// TIA Portal V17 export
// export: Created 2025-03-07T09:18:23.4469488Z, ExportSetting WithDefaults, DisplayName Totally Integrated Automation Portal, DisplayVersion V17 Update 8, DisplayName TIA Portal Openness, DisplayVersion V17 Update 8, DisplayName TIA Portal Version Control Interface, DisplayVersion V17, DisplayName SINAMICS Startdrive Advanced, DisplayVersion V17 SP2, DisplayName SINAMICS Startdrive G110M, G120, G120C, G120D, G120P, G115D, DisplayVersion V17 SP2, DisplayName SINAMICS Startdrive G130, G150, S120, S150, SINAMICS MV, S210, DisplayVersion V17 SP2, DisplayName STEP 7 Professional, DisplayVersion V17 Update 8, DisplayName SINUMERIK ONE STEP 7 Toolbox, DisplayVersion V17 Update 12, DisplayName SINUMERIK 840D sl STEP 7 Toolbox, DisplayVersion V17 Update 12, DisplayName STEP 7 Safety, DisplayVersion V17 Update 6, DisplayName WinCC Advanced, DisplayVersion V17 Update 8
FUNCTION_BLOCK "FB1453_LASER_COOLING_ALARMS"   // FB1453, LAD
{ S7_Optimized_Access := 'FALSE' }
AUTHOR : ETXETAR
VERSION : 1.0
// stored: AutoNumber false, IsIECCheckEnabled false, SetENOAutomatically false, UDAEnableTagReadback false
   VAR_INPUT
      OPTIONS_0 : Byte := 2#0000_0000;   // OPTIONS 0
      OPTIONS_1 : Byte := 2#0000_0000;   // OPTIONS 1
      LASER_OUTPUT_FLOW_LOW_VALUE_ALM_BIT : Bool;   // LASER OUTPUT FLOW LOW LEVEL ALARM BIT INPUT
      NOZZLE_FLOW_LOW_VALUE_ALM_BIT : Bool;   // NOZZLE FLOW LOW LEVEL ALARM BIT INPUT
      HEAD_FLOW_LOW_VALUE_ALM_BIT : Bool;   // HEAD FLOW LOW LEVEL ALARM BIT INPUT
      LASER_OUTPUT_OVERTEMPERATURE_ALM_BIT : Bool;   // LASER OUTPUT OVERTEMPERATURE ALARM BIT INPUT
      NOZZLE_OVERTEMPERATURE_ALM_BIT : Bool;   // NOZZLE OVERTEMPERATURE ALARM BIT INPUT
      HEAD_OVERTEMPERATURE_ALM_BIT : Bool;   // HEAD OVERTEMPERATURE ALARM BIT INPUT
      LASER_OUTPUT_FLOW_RAW_INPUT : DInt;   // LASER OUTPUT FLOW RAW INPUT
      LASER_OUTPUT_TEMP_RAW_INPUT : DInt;   // LASER OUTPUT TEMPERATURE RAW INPUT
      NOZZLE_COOLING_FLOW_RAW_INPUT : Word;   // NOZZLE FLOW RAW INPUT
      NOZZLE_COOLING_TEMP_RAW_INPUT : Word;   // NOOZLE TEMPERATURE RAW INPUT
      HEAD_COOLING_FLOW_RAW_INPUT : DInt;   // HEAD FLOW RAW INPUT
      HEAD_COOLING_TEMP_RAW_INPUT : DInt;   // HEAD TEMPERATURE RAW INPUT
      LASER_READY : Bool;   // THE LASER DEVICE IS READY
      UNIT_ALARM : UInt;   // UNIT NUMBER MAX. NUMBER=10
   END_VAR
   VAR_OUTPUT
      OUTPUT_LOW_FLOW_ALARM : Bool;   // LASER OUTPUT COOLING LOW FLOW ALARM
      OUTPUT_HIGH_FLOW_ALARM : Bool;   // LASER OUTPUT COOLING HIGH FLOW ALARM
      OUTPUT_FLOW_SETPOINT_ALARM : Bool;   // LASER OUTPUT COOLING FLOW SETPOINT ALARM
      OUTPUT_LOW_TEMP_ALARM : Bool;   // LASER OUTPUT COOLING LOW TEMPERATURE ALARM
      OUTPUT_HIGH_TEMP_ALARM : Bool;   // LASER OUTPUT COOLING HIGH TEMPERATURE ALARM
      OUTPUT_TEMP_SETPOINT_ALARM : Bool;   // LASER OUTPUT COOLING TEMPERATURE SETPOINT ALARM
      NOZZLE_LOW_FLOW_ALARM : Bool;   // NOZZLE COOLING LOW FLOW ALARM
      NOZZLE_HIGH_FLOW_ALARM : Bool;   // NOZZLE COOLING HIGH FLOW ALARM
      NOZZLE_FLOW_SETPOINT_ALARM : Bool;   // NOZZLE COOLING FLOW SETPOINT ALARM
      NOZZLE_LOW_TEMP_ALARM : Bool;   // NOZZLE COOLING LOW TEMPERATURE ALARM
      NOZZLE_HIGH_TEMP_ALARM : Bool;   // NOZZLE COOLING HIGH TEMPERATURE ALARM
      NOZZLE_TEMP_SETPOINT_ALARM : Bool;   // NOZZLE COOLING TEMPERATURE SETPOINT ALARM
      HEAD_LOW_FLOW_ALARM : Bool;   // LASER HEAD COOLING LOW FLOW ALARM
      HEAD_HIGH_FLOW_ALARM : Bool;   // LASER HEAD COOLING HIGH FLOW ALARM
      HEAD_FLOW_SETPOINT_ALARM : Bool;   // LASER HEAD COOLING FLOW SETPOINT ALARM
      HEAD_LOW_TEMP_ALARM : Bool;   // LASER HEAD COOLING LOW TEMPERATURE ALARM
      HEAD_HIGH_TEMP_ALARM : Bool;   // LASER HEAD COOLING HIGH TEMPERATURE ALARM
      HEAD_TEMP_SETPOINT_ALARM : Bool;   // LASER HEAD COOLING TEMPERATURE SETPOINT ALARM
      OUTPUT_LOW_FLOW_WARNING : Bool;   // LASER OUTPUT COOLING LOW FLOW WARNING
      OUTPUT_HIGH_FLOW_WARNING : Bool;   // LASER OUTPUT COOLING HIGH FLOW WARNING
      OUTPUT_LOW_TEMP_WARNING : Bool;   // LASER OUTPUT COOLING LOW TEMPERATURE WARNING
      OUTPUT_HIGH_TEMP_WARNING : Bool;   // LASER OUTPUT COOLING HIGH TEMPERATURE WARNING
      NOZZLE_LOW_FLOW_WARNING : Bool;   // NOZZLE COOLING LOW FLOW WARNING
      NOZZLE_HIGH_FLOW_WARNING : Bool;   // NOZZLE COOLING HIGH FLOW WARNING
      NOZZLE_LOW_TEMP_WARNING : Bool;   // NOZZLE COOLING LOW TEMPERATURE WARNING
      NOZZLE_HIGH_TEMP_WARNING : Bool;   // NOZZLE COOLING HIGH TEMPERATURE WARNING
      HEAD_LOW_FLOW_WARNING : Bool;   // LASER HEAD COOLING LOW FLOW WARNING
      HEAD_HIGH_FLOW_WARNING : Bool;   // LASER HEAD COOLING HIGH FLOW WARNING
      HEAD_LOW_TEMP_WARNING : Bool;   // LASER HEAD COOLING LOW TEMPERATURE WARNING
      HEAD_HIGH_TEMP_WARNING : Bool;   // LASER HEAD COOLING HIGH TEMPERATURE WARNING
   END_VAR
   VAR DB_SPECIFIC
      ANY_ACTIVE_ALARM : Bool;   // ANY ACTIVE ALARM
      RHP_SEOC_ALARMS : Bool;   // RETURN HOME POSITION AND STOP END OF CYCLE ALARMS
      IS_SEOC_ALARMS : Bool;   // INMEDIATE STOP AND STOP END OF CYCLE ALARMS
      WARNINGS : Bool;   // WARNINGS
      WARNINGS_GONE : Bool;   // WARNINGS GONE
      COOLING_ALARMS_ENABLED : Bool;   // COOLING ALARMS ENABLED
      LASER_OUTPUT_SENSOR_VALUES { ExternalAccessible := 'False'; ExternalVisible := 'False'; ExternalWritable := 'False'} : "COOLING_SENSOR";
      NOZZLE_SENSOR_VALUES { ExternalAccessible := 'False'; ExternalVisible := 'False'; ExternalWritable := 'False'} : "COOLING_SENSOR";
      LASER_HEAD_SENSOR_VALUES { ExternalAccessible := 'False'; ExternalVisible := 'False'; ExternalWritable := 'False'} : "COOLING_SENSOR";
   END_VAR
   VAR_TEMP
      INPUTS_MASK : Byte;   // INPUT MASK
      O_BYTE_0 : Struct   // OPTIONS BYTE 0
         OUTPUT_FLOW_LOW_BIT_ALARM : Bool;   // CIRCUIT BREAKER OPTION
         NOZZLE_FLOW_LOW_BIT_ALARM : Bool;   // CONTACTOR FEEDBACK OPTION
         HEAD_FLOW_LOW_BIT_ALARM : Bool;   // LOW LEVEL ALARM OPTION
         OUTPUT_FLOW_ANALOG_VALUE : Bool;   // SYSTEM ALARM 1 OPTION
         NOZZLE_FLOW_ANALOG_VALUE : Bool;   // SYSTEM ALARM 2 OPTION
         HEAD_FLOW_ANALOG_VALUE : Bool;   // FILTER CLOGGED ALARM OPTION
         SPARE_6 : Bool;   // OVERTEMPERATURE ALARM OPTION
         SPARE_7 : Bool;   // WATER SUPPLY FLOW OPTION
      END_STRUCT;
      O_BYTE_1 : Struct   // OPTIONS BYTE 1
         OUTPUT_TEMP_HIGH_BIT_ALARM : Bool;   // LOW LEVEL PREALARM OPTION
         NOZZLE_TEMP_HIGH_BIT_ALARM : Bool;   // FILTER CLOGGED PREALARM OPTION
         HEAD_TEMP_HIGH_BIT_ALARM : Bool;   // OVERTEMPERATURE PREALARM OPTION
         OUTPUT_TEMP_ANALOG_VALUE : Bool;   // DIGITAL FLOW SENSORS OPTION
         NOZZLE_TEMP_ANALOG_VALUE : Bool;   // SPARE OPTION
         HEAD_TEMP_ANALOG_VALUE : Bool;   // SPARE OPTION
         SPARE_6 : Bool;   // SPARE OPTION
         SPARE_7 : Bool;   // SPARE OPTION
      END_STRUCT;
      DB_NUMBER : DInt;   // DB NUMBER FOR ALARM AND HELP DECODING
      COOLING_TEMP_AUX_OUTPUT : Real;   // COOLING OUTPUT TEMPERATURE AUX
      COOLING_FLOW_AUX_OUTPUT : Real;   // COOLING OUTPUT FLOW AUX
      COOLING_TEMP_AUX_3 : Int;   // COOLING TEMPERATURE AUX 3
   END_VAR
   VAR_TEMP   // added for the SCL form of the ladder/FBD networks
      _w1 : Bool;
   END_VAR
BEGIN

NETWORK
TITLE = READ INSTANCE DB
      L     DINO;
      +     10#800000;
      T     #DB_NUMBER;


REGION Network 2: OPTIONS
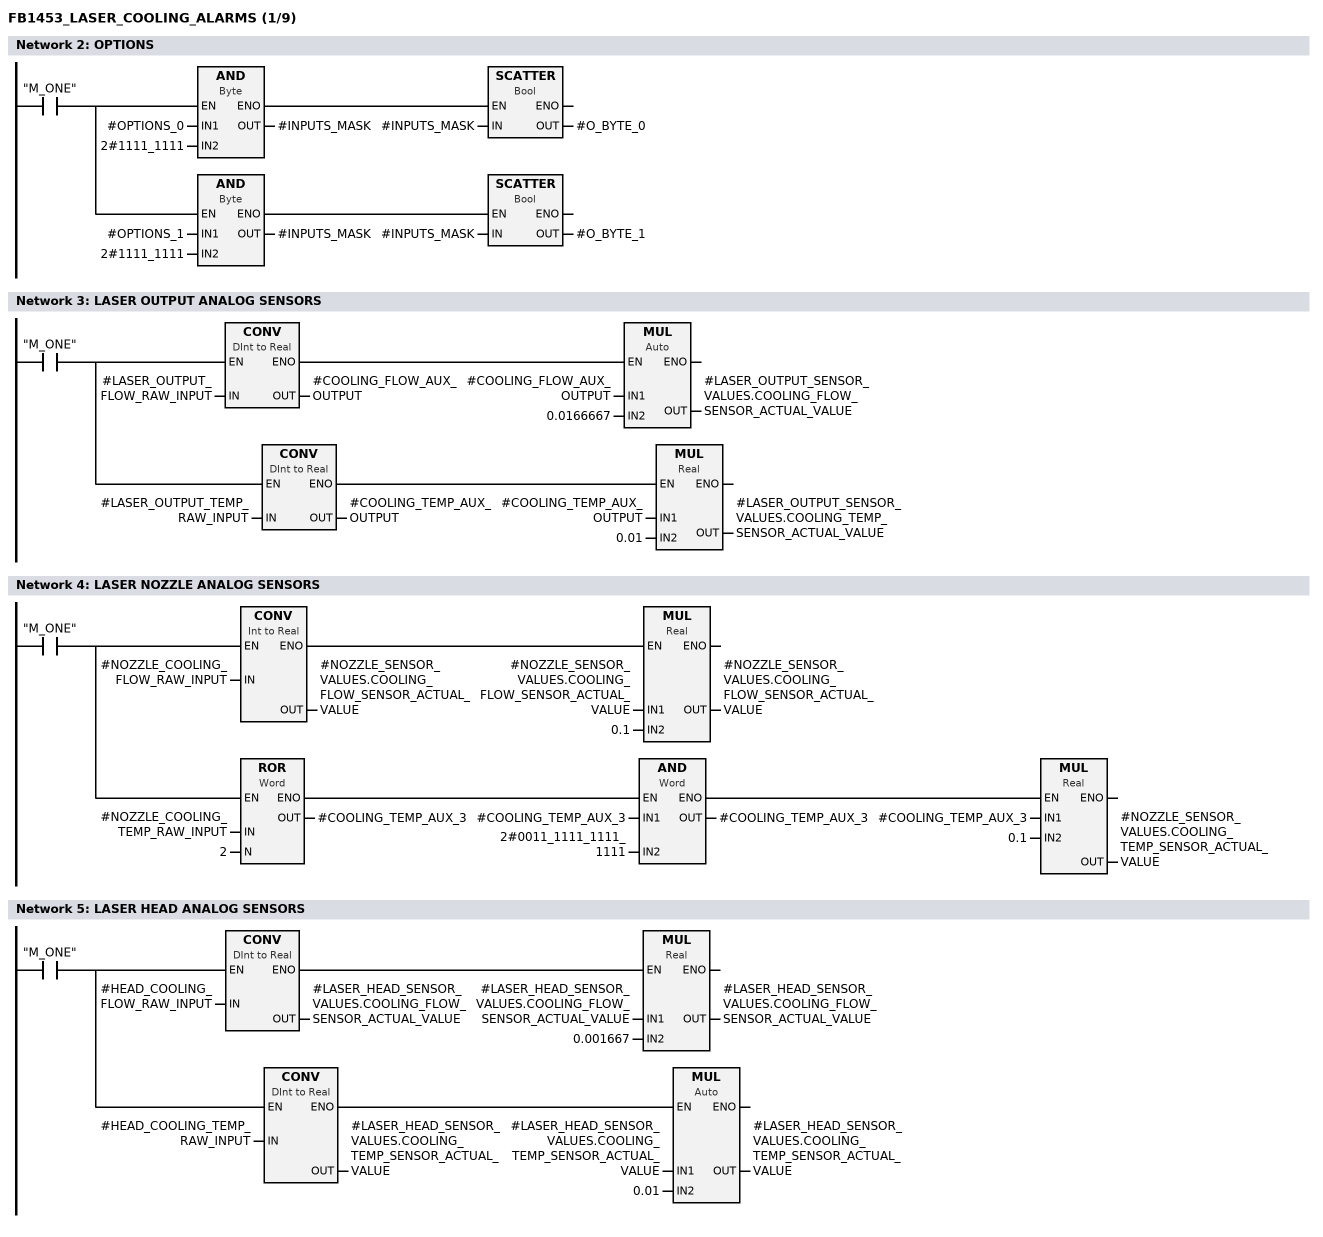
   RUNG wire#powerrail
      Contact( "M_ONE" )
      wire#w1
      { S7_Templates := "SrcType := Byte"; S7_GenerateENO := "TRUE" } And(in1 := #OPTIONS_0, in2 := 2#1111_1111, out => #INPUTS_MASK)
      { S7_Templates := "[dest_type := Bool, src_type := Byte]" } SCATTER(IN := #INPUTS_MASK, OUT => #O_BYTE_0)
   END_RUNG
   RUNG wire#w1
      { S7_Templates := "SrcType := Byte"; S7_GenerateENO := "TRUE" } And(in1 := #OPTIONS_1, in2 := 2#1111_1111, out => #INPUTS_MASK)
      { S7_Templates := "[dest_type := Bool, src_type := Byte]" } SCATTER(IN := #INPUTS_MASK, OUT => #O_BYTE_1)
   END_RUNG
   // the same network as SCL:
   IF "M_ONE" THEN #INPUTS_MASK := #OPTIONS_0 AND 2#1111_1111; END_IF;
   #_w1 := "M_ONE";
   IF #_w1 THEN
       SCATTER(IN := #INPUTS_MASK, OUT => #O_BYTE_0);
       #INPUTS_MASK := #OPTIONS_1 AND 2#1111_1111;
       SCATTER(IN := #INPUTS_MASK, OUT => #O_BYTE_1);
   END_IF;
END_REGION

REGION Network 3: LASER OUTPUT ANALOG SENSORS
   RUNG wire#powerrail
      Contact( "M_ONE" )
      wire#w1
      { S7_Templates := "[SrcType := DInt, DestType := Real]" } Convert(in := #LASER_OUTPUT_FLOW_RAW_INPUT, out => #COOLING_FLOW_AUX_OUTPUT)
      Mul(in1 := #COOLING_FLOW_AUX_OUTPUT, in2 := 0.0166667, out => #LASER_OUTPUT_SENSOR_VALUES.COOLING_FLOW_SENSOR_ACTUAL_VALUE)
   END_RUNG
   RUNG wire#w1
      { S7_Templates := "[SrcType := DInt, DestType := Real]" } Convert(in := #LASER_OUTPUT_TEMP_RAW_INPUT, out => #COOLING_TEMP_AUX_OUTPUT)
      { S7_Templates := "SrcType := Real" } Mul(in1 := #COOLING_TEMP_AUX_OUTPUT, in2 := 0.01, out => #LASER_OUTPUT_SENSOR_VALUES.COOLING_TEMP_SENSOR_ACTUAL_VALUE)
   END_RUNG
   // the same network as SCL:
   IF "M_ONE" THEN
       #COOLING_FLOW_AUX_OUTPUT := DINT_TO_REAL(#LASER_OUTPUT_FLOW_RAW_INPUT);
       #LASER_OUTPUT_SENSOR_VALUES.COOLING_FLOW_SENSOR_ACTUAL_VALUE := #COOLING_FLOW_AUX_OUTPUT * 0.0166667;
       #COOLING_TEMP_AUX_OUTPUT := DINT_TO_REAL(#LASER_OUTPUT_TEMP_RAW_INPUT);
       #LASER_OUTPUT_SENSOR_VALUES.COOLING_TEMP_SENSOR_ACTUAL_VALUE := #COOLING_TEMP_AUX_OUTPUT * 0.01;
   END_IF;
END_REGION

REGION Network 4: LASER NOZZLE ANALOG SENSORS
   IF "M_ONE" THEN
       #NOZZLE_SENSOR_VALUES.COOLING_FLOW_SENSOR_ACTUAL_VALUE := INT_TO_REAL(#NOZZLE_COOLING_FLOW_RAW_INPUT);
       #NOZZLE_SENSOR_VALUES.COOLING_FLOW_SENSOR_ACTUAL_VALUE := #NOZZLE_SENSOR_VALUES.COOLING_FLOW_SENSOR_ACTUAL_VALUE * 0.1;
       #COOLING_TEMP_AUX_3 := ROR(IN := #NOZZLE_COOLING_TEMP_RAW_INPUT, N := 2);
       #COOLING_TEMP_AUX_3 := #COOLING_TEMP_AUX_3 AND 2#0011_1111_1111_1111;
       #NOZZLE_SENSOR_VALUES.COOLING_TEMP_SENSOR_ACTUAL_VALUE := #COOLING_TEMP_AUX_3 * 0.1;
   END_IF;
END_REGION

REGION Network 5: LASER HEAD ANALOG SENSORS
   RUNG wire#powerrail
      Contact( "M_ONE" )
      wire#w1
      { S7_Templates := "[SrcType := DInt, DestType := Real]" } Convert(in := #HEAD_COOLING_FLOW_RAW_INPUT, out => #LASER_HEAD_SENSOR_VALUES.COOLING_FLOW_SENSOR_ACTUAL_VALUE)
      { S7_Templates := "SrcType := Real" } Mul(in1 := #LASER_HEAD_SENSOR_VALUES.COOLING_FLOW_SENSOR_ACTUAL_VALUE, in2 := 0.001667, out => #LASER_HEAD_SENSOR_VALUES.COOLING_FLOW_SENSOR_ACTUAL_VALUE)
   END_RUNG
   RUNG wire#w1
      { S7_Templates := "[SrcType := DInt, DestType := Real]"; S7_GenerateENO := "TRUE" } Convert(in := #HEAD_COOLING_TEMP_RAW_INPUT, out => #LASER_HEAD_SENSOR_VALUES.COOLING_TEMP_SENSOR_ACTUAL_VALUE)
      { S7_GenerateENO := "TRUE" } Mul(in1 := #LASER_HEAD_SENSOR_VALUES.COOLING_TEMP_SENSOR_ACTUAL_VALUE, in2 := 0.01, out => #LASER_HEAD_SENSOR_VALUES.COOLING_TEMP_SENSOR_ACTUAL_VALUE)
   END_RUNG
   // the same network as SCL:
   // ENO of a box is taken as its EN; it also drops when the box reports an error
   IF "M_ONE" THEN
       #LASER_HEAD_SENSOR_VALUES.COOLING_FLOW_SENSOR_ACTUAL_VALUE := DINT_TO_REAL(#HEAD_COOLING_FLOW_RAW_INPUT);
       #LASER_HEAD_SENSOR_VALUES.COOLING_FLOW_SENSOR_ACTUAL_VALUE := #LASER_HEAD_SENSOR_VALUES.COOLING_FLOW_SENSOR_ACTUAL_VALUE * 0.001667;
       #LASER_HEAD_SENSOR_VALUES.COOLING_TEMP_SENSOR_ACTUAL_VALUE := DINT_TO_REAL(#HEAD_COOLING_TEMP_RAW_INPUT);
       #LASER_HEAD_SENSOR_VALUES.COOLING_TEMP_SENSOR_ACTUAL_VALUE := #LASER_HEAD_SENSOR_VALUES.COOLING_TEMP_SENSOR_ACTUAL_VALUE * 0.01;
   END_IF;
END_REGION

REGION Network 6: COOLING SENSOR LASER OUTPUT FLOW WARNINGS/ALARMS
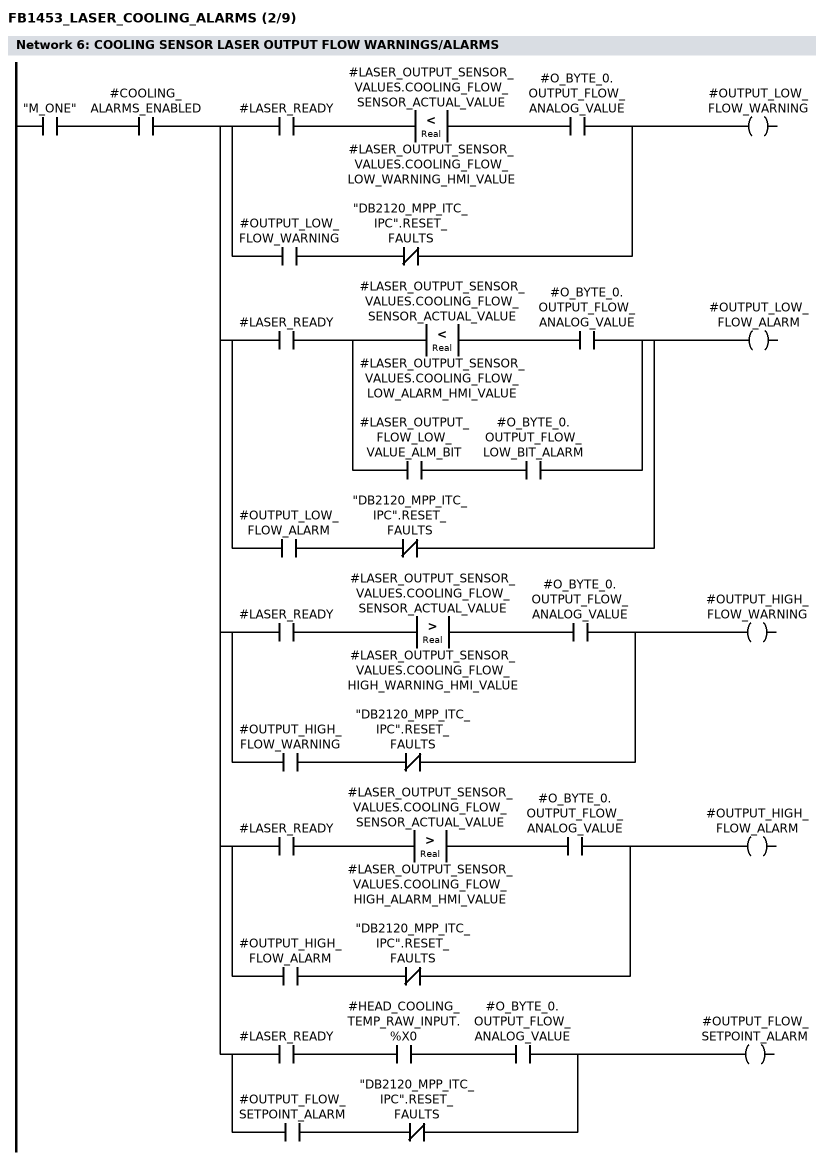
   RUNG wire#powerrail
      Contact( "M_ONE" )
      Contact( #COOLING_ALARMS_ENABLED )
      wire#w1
      Contact( #LASER_READY )
      { S7_Templates := "SrcType := Real" } LT_Contact(in1 := #LASER_OUTPUT_SENSOR_VALUES.COOLING_FLOW_SENSOR_ACTUAL_VALUE, in2 := #LASER_OUTPUT_SENSOR_VALUES.COOLING_FLOW_LOW_WARNING_HMI_VALUE)
      Contact( #O_BYTE_0.OUTPUT_FLOW_ANALOG_VALUE )
      wire#w2
      Coil( #OUTPUT_LOW_FLOW_WARNING )
   END_RUNG
   RUNG wire#w1
      Contact( #OUTPUT_LOW_FLOW_WARNING )
      I_Contact( "DB2120_MPP_ITC_IPC".RESET_FAULTS )
   END_RUNG wire#w2
   RUNG wire#w1
      Contact( #LASER_READY )
      wire#w3
      { S7_Templates := "SrcType := Real" } LT_Contact(in1 := #LASER_OUTPUT_SENSOR_VALUES.COOLING_FLOW_SENSOR_ACTUAL_VALUE, in2 := #LASER_OUTPUT_SENSOR_VALUES.COOLING_FLOW_LOW_ALARM_HMI_VALUE)
      Contact( #O_BYTE_0.OUTPUT_FLOW_ANALOG_VALUE )
      wire#w4
      Coil( #OUTPUT_LOW_FLOW_ALARM )
   END_RUNG
   RUNG wire#w3
      Contact( #LASER_OUTPUT_FLOW_LOW_VALUE_ALM_BIT )
      Contact( #O_BYTE_0.OUTPUT_FLOW_LOW_BIT_ALARM )
   END_RUNG wire#w4
   RUNG wire#w1
      Contact( #OUTPUT_LOW_FLOW_ALARM )
      I_Contact( "DB2120_MPP_ITC_IPC".RESET_FAULTS )
   END_RUNG wire#w4
   RUNG wire#w1
      Contact( #LASER_READY )
      { S7_Templates := "SrcType := Real" } GT_Contact(in1 := #LASER_OUTPUT_SENSOR_VALUES.COOLING_FLOW_SENSOR_ACTUAL_VALUE, in2 := #LASER_OUTPUT_SENSOR_VALUES.COOLING_FLOW_HIGH_WARNING_HMI_VALUE)
      Contact( #O_BYTE_0.OUTPUT_FLOW_ANALOG_VALUE )
      wire#w5
      Coil( #OUTPUT_HIGH_FLOW_WARNING )
   END_RUNG
   RUNG wire#w1
      Contact( #OUTPUT_HIGH_FLOW_WARNING )
      I_Contact( "DB2120_MPP_ITC_IPC".RESET_FAULTS )
   END_RUNG wire#w5
   RUNG wire#w1
      Contact( #LASER_READY )
      { S7_Templates := "SrcType := Real" } GT_Contact(in1 := #LASER_OUTPUT_SENSOR_VALUES.COOLING_FLOW_SENSOR_ACTUAL_VALUE, in2 := #LASER_OUTPUT_SENSOR_VALUES.COOLING_FLOW_HIGH_ALARM_HMI_VALUE)
      Contact( #O_BYTE_0.OUTPUT_FLOW_ANALOG_VALUE )
      wire#w6
      Coil( #OUTPUT_HIGH_FLOW_ALARM )
   END_RUNG
   RUNG wire#w1
      Contact( #OUTPUT_HIGH_FLOW_ALARM )
      I_Contact( "DB2120_MPP_ITC_IPC".RESET_FAULTS )
   END_RUNG wire#w6
   RUNG wire#w1
      Contact( #LASER_READY )
      Contact( #HEAD_COOLING_TEMP_RAW_INPUT.%X0 )
      Contact( #O_BYTE_0.OUTPUT_FLOW_ANALOG_VALUE )
      wire#w7
      Coil( #OUTPUT_FLOW_SETPOINT_ALARM )
   END_RUNG
   RUNG wire#w1
      Contact( #OUTPUT_FLOW_SETPOINT_ALARM )
      I_Contact( "DB2120_MPP_ITC_IPC".RESET_FAULTS )
   END_RUNG wire#w7
   // the same network as SCL:
   #_w1 := "M_ONE" AND #COOLING_ALARMS_ENABLED;
   #OUTPUT_LOW_FLOW_WARNING := #_w1 AND ((#LASER_READY AND (#LASER_OUTPUT_SENSOR_VALUES.COOLING_FLOW_SENSOR_ACTUAL_VALUE < #LASER_OUTPUT_SENSOR_VALUES.COOLING_FLOW_LOW_WARNING_HMI_VALUE) AND #O_BYTE_0.OUTPUT_FLOW_ANALOG_VALUE) OR (#OUTPUT_LOW_FLOW_WARNING AND NOT "DB2120_MPP_ITC_IPC".RESET_FAULTS));
   #OUTPUT_LOW_FLOW_ALARM := #_w1 AND ((#LASER_READY AND (((#LASER_OUTPUT_SENSOR_VALUES.COOLING_FLOW_SENSOR_ACTUAL_VALUE < #LASER_OUTPUT_SENSOR_VALUES.COOLING_FLOW_LOW_ALARM_HMI_VALUE) AND #O_BYTE_0.OUTPUT_FLOW_ANALOG_VALUE) OR (#LASER_OUTPUT_FLOW_LOW_VALUE_ALM_BIT AND #O_BYTE_0.OUTPUT_FLOW_LOW_BIT_ALARM))) OR (#OUTPUT_LOW_FLOW_ALARM AND NOT "DB2120_MPP_ITC_IPC".RESET_FAULTS));
   #OUTPUT_HIGH_FLOW_WARNING := #_w1 AND ((#LASER_READY AND (#LASER_OUTPUT_SENSOR_VALUES.COOLING_FLOW_SENSOR_ACTUAL_VALUE > #LASER_OUTPUT_SENSOR_VALUES.COOLING_FLOW_HIGH_WARNING_HMI_VALUE) AND #O_BYTE_0.OUTPUT_FLOW_ANALOG_VALUE) OR (#OUTPUT_HIGH_FLOW_WARNING AND NOT "DB2120_MPP_ITC_IPC".RESET_FAULTS));
   #OUTPUT_HIGH_FLOW_ALARM := #_w1 AND ((#LASER_READY AND (#LASER_OUTPUT_SENSOR_VALUES.COOLING_FLOW_SENSOR_ACTUAL_VALUE > #LASER_OUTPUT_SENSOR_VALUES.COOLING_FLOW_HIGH_ALARM_HMI_VALUE) AND #O_BYTE_0.OUTPUT_FLOW_ANALOG_VALUE) OR (#OUTPUT_HIGH_FLOW_ALARM AND NOT "DB2120_MPP_ITC_IPC".RESET_FAULTS));
   #OUTPUT_FLOW_SETPOINT_ALARM := #_w1 AND ((#LASER_READY AND #HEAD_COOLING_TEMP_RAW_INPUT.%X0 AND #O_BYTE_0.OUTPUT_FLOW_ANALOG_VALUE) OR (#OUTPUT_FLOW_SETPOINT_ALARM AND NOT "DB2120_MPP_ITC_IPC".RESET_FAULTS));
END_REGION

REGION Network 7: COOLING SENSOR LASER OUTPUT TEMPERATURE WARNINGS/ALARMS
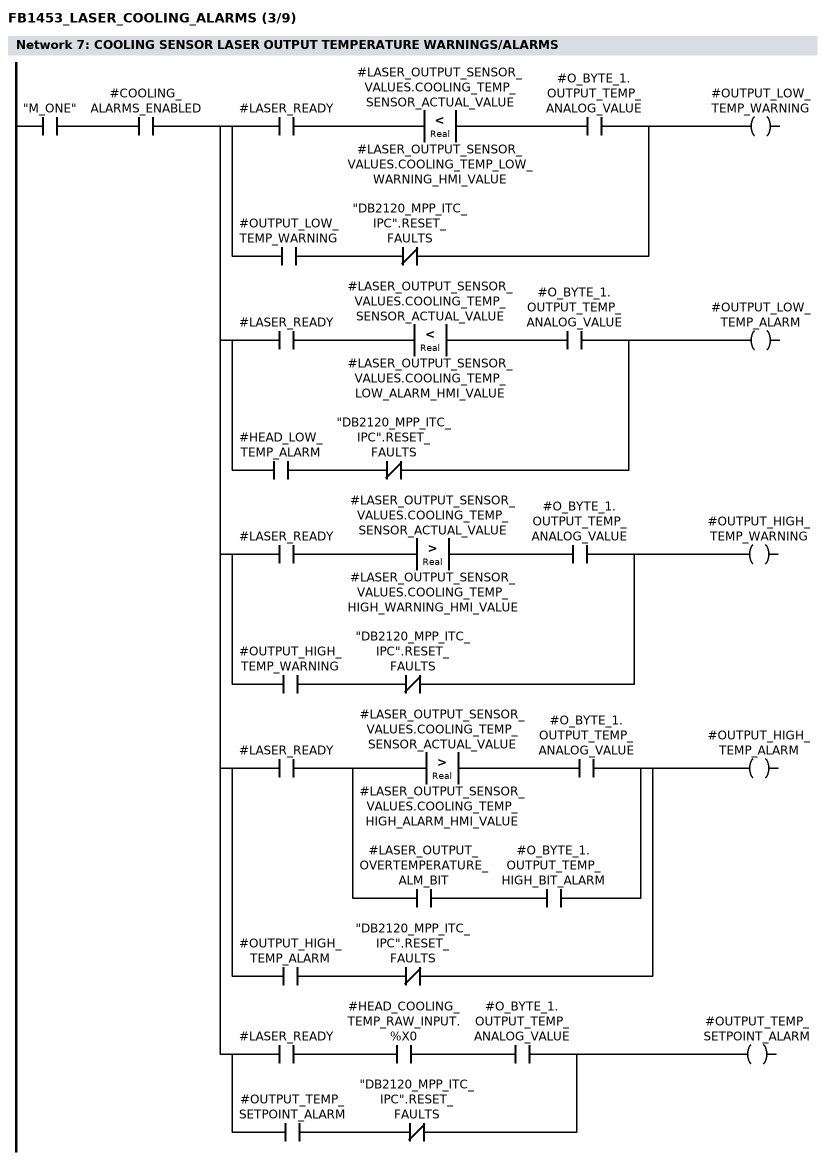
   RUNG wire#powerrail
      Contact( "M_ONE" )
      Contact( #COOLING_ALARMS_ENABLED )
      wire#w1
      Contact( #LASER_READY )
      { S7_Templates := "SrcType := Real" } LT_Contact(in1 := #LASER_OUTPUT_SENSOR_VALUES.COOLING_TEMP_SENSOR_ACTUAL_VALUE, in2 := #LASER_OUTPUT_SENSOR_VALUES.COOLING_TEMP_LOW_WARNING_HMI_VALUE)
      Contact( #O_BYTE_1.OUTPUT_TEMP_ANALOG_VALUE )
      wire#w2
      Coil( #OUTPUT_LOW_TEMP_WARNING )
   END_RUNG
   RUNG wire#w1
      Contact( #OUTPUT_LOW_TEMP_WARNING )
      I_Contact( "DB2120_MPP_ITC_IPC".RESET_FAULTS )
   END_RUNG wire#w2
   RUNG wire#w1
      Contact( #LASER_READY )
      { S7_Templates := "SrcType := Real" } LT_Contact(in1 := #LASER_OUTPUT_SENSOR_VALUES.COOLING_TEMP_SENSOR_ACTUAL_VALUE, in2 := #LASER_OUTPUT_SENSOR_VALUES.COOLING_TEMP_LOW_ALARM_HMI_VALUE)
      Contact( #O_BYTE_1.OUTPUT_TEMP_ANALOG_VALUE )
      wire#w3
      Coil( #OUTPUT_LOW_TEMP_ALARM )
   END_RUNG
   RUNG wire#w1
      Contact( #HEAD_LOW_TEMP_ALARM )
      I_Contact( "DB2120_MPP_ITC_IPC".RESET_FAULTS )
   END_RUNG wire#w3
   RUNG wire#w1
      Contact( #LASER_READY )
      { S7_Templates := "SrcType := Real" } GT_Contact(in1 := #LASER_OUTPUT_SENSOR_VALUES.COOLING_TEMP_SENSOR_ACTUAL_VALUE, in2 := #LASER_OUTPUT_SENSOR_VALUES.COOLING_TEMP_HIGH_WARNING_HMI_VALUE)
      Contact( #O_BYTE_1.OUTPUT_TEMP_ANALOG_VALUE )
      wire#w4
      Coil( #OUTPUT_HIGH_TEMP_WARNING )
   END_RUNG
   RUNG wire#w1
      Contact( #OUTPUT_HIGH_TEMP_WARNING )
      I_Contact( "DB2120_MPP_ITC_IPC".RESET_FAULTS )
   END_RUNG wire#w4
   RUNG wire#w1
      Contact( #LASER_READY )
      wire#w5
      { S7_Templates := "SrcType := Real" } GT_Contact(in1 := #LASER_OUTPUT_SENSOR_VALUES.COOLING_TEMP_SENSOR_ACTUAL_VALUE, in2 := #LASER_OUTPUT_SENSOR_VALUES.COOLING_TEMP_HIGH_ALARM_HMI_VALUE)
      Contact( #O_BYTE_1.OUTPUT_TEMP_ANALOG_VALUE )
      wire#w6
      Coil( #OUTPUT_HIGH_TEMP_ALARM )
   END_RUNG
   RUNG wire#w5
      Contact( #LASER_OUTPUT_OVERTEMPERATURE_ALM_BIT )
      Contact( #O_BYTE_1.OUTPUT_TEMP_HIGH_BIT_ALARM )
   END_RUNG wire#w6
   RUNG wire#w1
      Contact( #OUTPUT_HIGH_TEMP_ALARM )
      I_Contact( "DB2120_MPP_ITC_IPC".RESET_FAULTS )
   END_RUNG wire#w6
   RUNG wire#w1
      Contact( #LASER_READY )
      Contact( #HEAD_COOLING_TEMP_RAW_INPUT.%X0 )
      Contact( #O_BYTE_1.OUTPUT_TEMP_ANALOG_VALUE )
      wire#w7
      Coil( #OUTPUT_TEMP_SETPOINT_ALARM )
   END_RUNG
   RUNG wire#w1
      Contact( #OUTPUT_TEMP_SETPOINT_ALARM )
      I_Contact( "DB2120_MPP_ITC_IPC".RESET_FAULTS )
   END_RUNG wire#w7
   // the same network as SCL:
   #_w1 := "M_ONE" AND #COOLING_ALARMS_ENABLED;
   #OUTPUT_LOW_TEMP_WARNING := #_w1 AND ((#LASER_READY AND (#LASER_OUTPUT_SENSOR_VALUES.COOLING_TEMP_SENSOR_ACTUAL_VALUE < #LASER_OUTPUT_SENSOR_VALUES.COOLING_TEMP_LOW_WARNING_HMI_VALUE) AND #O_BYTE_1.OUTPUT_TEMP_ANALOG_VALUE) OR (#OUTPUT_LOW_TEMP_WARNING AND NOT "DB2120_MPP_ITC_IPC".RESET_FAULTS));
   #OUTPUT_LOW_TEMP_ALARM := #_w1 AND ((#LASER_READY AND (#LASER_OUTPUT_SENSOR_VALUES.COOLING_TEMP_SENSOR_ACTUAL_VALUE < #LASER_OUTPUT_SENSOR_VALUES.COOLING_TEMP_LOW_ALARM_HMI_VALUE) AND #O_BYTE_1.OUTPUT_TEMP_ANALOG_VALUE) OR (#HEAD_LOW_TEMP_ALARM AND NOT "DB2120_MPP_ITC_IPC".RESET_FAULTS));
   #OUTPUT_HIGH_TEMP_WARNING := #_w1 AND ((#LASER_READY AND (#LASER_OUTPUT_SENSOR_VALUES.COOLING_TEMP_SENSOR_ACTUAL_VALUE > #LASER_OUTPUT_SENSOR_VALUES.COOLING_TEMP_HIGH_WARNING_HMI_VALUE) AND #O_BYTE_1.OUTPUT_TEMP_ANALOG_VALUE) OR (#OUTPUT_HIGH_TEMP_WARNING AND NOT "DB2120_MPP_ITC_IPC".RESET_FAULTS));
   #OUTPUT_HIGH_TEMP_ALARM := #_w1 AND ((#LASER_READY AND (((#LASER_OUTPUT_SENSOR_VALUES.COOLING_TEMP_SENSOR_ACTUAL_VALUE > #LASER_OUTPUT_SENSOR_VALUES.COOLING_TEMP_HIGH_ALARM_HMI_VALUE) AND #O_BYTE_1.OUTPUT_TEMP_ANALOG_VALUE) OR (#LASER_OUTPUT_OVERTEMPERATURE_ALM_BIT AND #O_BYTE_1.OUTPUT_TEMP_HIGH_BIT_ALARM))) OR (#OUTPUT_HIGH_TEMP_ALARM AND NOT "DB2120_MPP_ITC_IPC".RESET_FAULTS));
   #OUTPUT_TEMP_SETPOINT_ALARM := #_w1 AND ((#LASER_READY AND #HEAD_COOLING_TEMP_RAW_INPUT.%X0 AND #O_BYTE_1.OUTPUT_TEMP_ANALOG_VALUE) OR (#OUTPUT_TEMP_SETPOINT_ALARM AND NOT "DB2120_MPP_ITC_IPC".RESET_FAULTS));
END_REGION

REGION Network 8: COOLING SENSOR NOZZLE FLOW WARNINGS/ALARMS
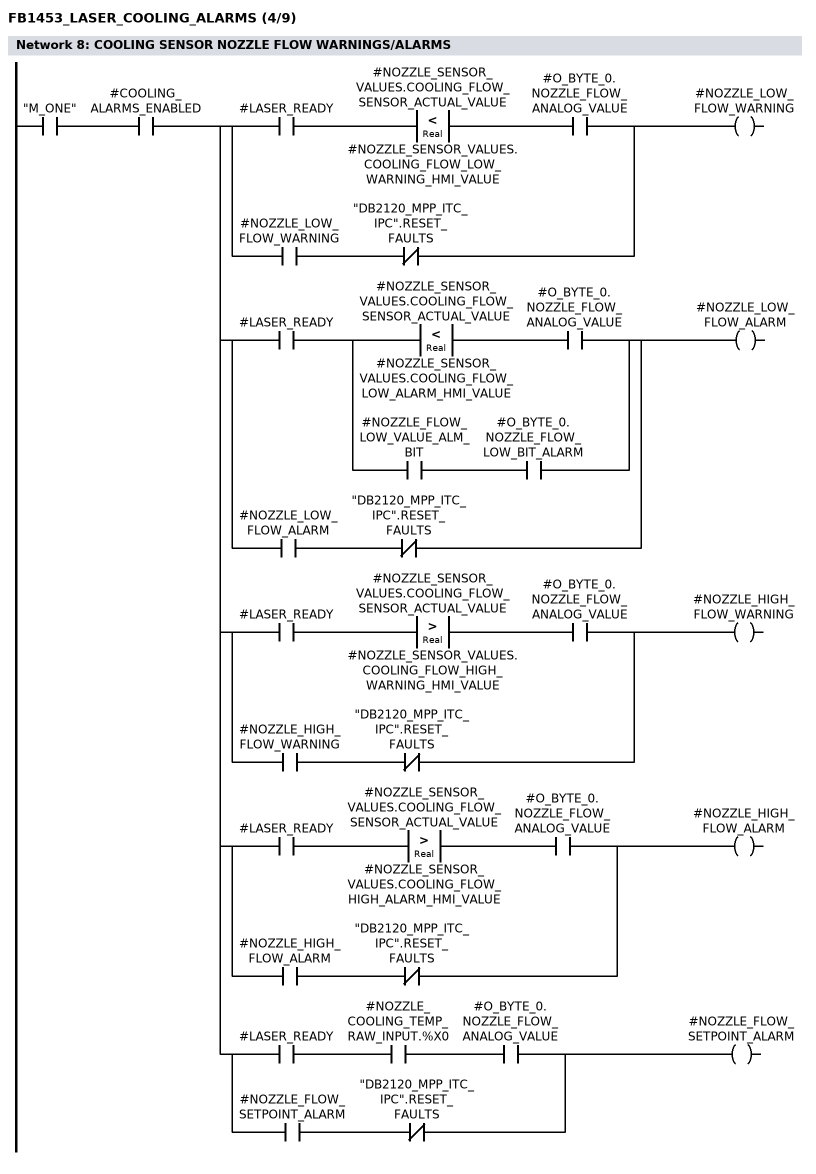
   RUNG wire#powerrail
      Contact( "M_ONE" )
      Contact( #COOLING_ALARMS_ENABLED )
      wire#w1
      Contact( #LASER_READY )
      { S7_Templates := "SrcType := Real" } LT_Contact(in1 := #NOZZLE_SENSOR_VALUES.COOLING_FLOW_SENSOR_ACTUAL_VALUE, in2 := #NOZZLE_SENSOR_VALUES.COOLING_FLOW_LOW_WARNING_HMI_VALUE)
      Contact( #O_BYTE_0.NOZZLE_FLOW_ANALOG_VALUE )
      wire#w2
      Coil( #NOZZLE_LOW_FLOW_WARNING )
   END_RUNG
   RUNG wire#w1
      Contact( #NOZZLE_LOW_FLOW_WARNING )
      I_Contact( "DB2120_MPP_ITC_IPC".RESET_FAULTS )
   END_RUNG wire#w2
   RUNG wire#w1
      Contact( #LASER_READY )
      wire#w3
      { S7_Templates := "SrcType := Real" } LT_Contact(in1 := #NOZZLE_SENSOR_VALUES.COOLING_FLOW_SENSOR_ACTUAL_VALUE, in2 := #NOZZLE_SENSOR_VALUES.COOLING_FLOW_LOW_ALARM_HMI_VALUE)
      Contact( #O_BYTE_0.NOZZLE_FLOW_ANALOG_VALUE )
      wire#w4
      Coil( #NOZZLE_LOW_FLOW_ALARM )
   END_RUNG
   RUNG wire#w3
      Contact( #NOZZLE_FLOW_LOW_VALUE_ALM_BIT )
      Contact( #O_BYTE_0.NOZZLE_FLOW_LOW_BIT_ALARM )
   END_RUNG wire#w4
   RUNG wire#w1
      Contact( #NOZZLE_LOW_FLOW_ALARM )
      I_Contact( "DB2120_MPP_ITC_IPC".RESET_FAULTS )
   END_RUNG wire#w4
   RUNG wire#w1
      Contact( #LASER_READY )
      { S7_Templates := "SrcType := Real" } GT_Contact(in1 := #NOZZLE_SENSOR_VALUES.COOLING_FLOW_SENSOR_ACTUAL_VALUE, in2 := #NOZZLE_SENSOR_VALUES.COOLING_FLOW_HIGH_WARNING_HMI_VALUE)
      Contact( #O_BYTE_0.NOZZLE_FLOW_ANALOG_VALUE )
      wire#w5
      Coil( #NOZZLE_HIGH_FLOW_WARNING )
   END_RUNG
   RUNG wire#w1
      Contact( #NOZZLE_HIGH_FLOW_WARNING )
      I_Contact( "DB2120_MPP_ITC_IPC".RESET_FAULTS )
   END_RUNG wire#w5
   RUNG wire#w1
      Contact( #LASER_READY )
      { S7_Templates := "SrcType := Real" } GT_Contact(in1 := #NOZZLE_SENSOR_VALUES.COOLING_FLOW_SENSOR_ACTUAL_VALUE, in2 := #NOZZLE_SENSOR_VALUES.COOLING_FLOW_HIGH_ALARM_HMI_VALUE)
      Contact( #O_BYTE_0.NOZZLE_FLOW_ANALOG_VALUE )
      wire#w6
      Coil( #NOZZLE_HIGH_FLOW_ALARM )
   END_RUNG
   RUNG wire#w1
      Contact( #NOZZLE_HIGH_FLOW_ALARM )
      I_Contact( "DB2120_MPP_ITC_IPC".RESET_FAULTS )
   END_RUNG wire#w6
   RUNG wire#w1
      Contact( #LASER_READY )
      Contact( #NOZZLE_COOLING_TEMP_RAW_INPUT.%X0 )
      Contact( #O_BYTE_0.NOZZLE_FLOW_ANALOG_VALUE )
      wire#w7
      Coil( #NOZZLE_FLOW_SETPOINT_ALARM )
   END_RUNG
   RUNG wire#w1
      Contact( #NOZZLE_FLOW_SETPOINT_ALARM )
      I_Contact( "DB2120_MPP_ITC_IPC".RESET_FAULTS )
   END_RUNG wire#w7
   // the same network as SCL:
   #_w1 := "M_ONE" AND #COOLING_ALARMS_ENABLED;
   #NOZZLE_LOW_FLOW_WARNING := #_w1 AND ((#LASER_READY AND (#NOZZLE_SENSOR_VALUES.COOLING_FLOW_SENSOR_ACTUAL_VALUE < #NOZZLE_SENSOR_VALUES.COOLING_FLOW_LOW_WARNING_HMI_VALUE) AND #O_BYTE_0.NOZZLE_FLOW_ANALOG_VALUE) OR (#NOZZLE_LOW_FLOW_WARNING AND NOT "DB2120_MPP_ITC_IPC".RESET_FAULTS));
   #NOZZLE_LOW_FLOW_ALARM := #_w1 AND ((#LASER_READY AND (((#NOZZLE_SENSOR_VALUES.COOLING_FLOW_SENSOR_ACTUAL_VALUE < #NOZZLE_SENSOR_VALUES.COOLING_FLOW_LOW_ALARM_HMI_VALUE) AND #O_BYTE_0.NOZZLE_FLOW_ANALOG_VALUE) OR (#NOZZLE_FLOW_LOW_VALUE_ALM_BIT AND #O_BYTE_0.NOZZLE_FLOW_LOW_BIT_ALARM))) OR (#NOZZLE_LOW_FLOW_ALARM AND NOT "DB2120_MPP_ITC_IPC".RESET_FAULTS));
   #NOZZLE_HIGH_FLOW_WARNING := #_w1 AND ((#LASER_READY AND (#NOZZLE_SENSOR_VALUES.COOLING_FLOW_SENSOR_ACTUAL_VALUE > #NOZZLE_SENSOR_VALUES.COOLING_FLOW_HIGH_WARNING_HMI_VALUE) AND #O_BYTE_0.NOZZLE_FLOW_ANALOG_VALUE) OR (#NOZZLE_HIGH_FLOW_WARNING AND NOT "DB2120_MPP_ITC_IPC".RESET_FAULTS));
   #NOZZLE_HIGH_FLOW_ALARM := #_w1 AND ((#LASER_READY AND (#NOZZLE_SENSOR_VALUES.COOLING_FLOW_SENSOR_ACTUAL_VALUE > #NOZZLE_SENSOR_VALUES.COOLING_FLOW_HIGH_ALARM_HMI_VALUE) AND #O_BYTE_0.NOZZLE_FLOW_ANALOG_VALUE) OR (#NOZZLE_HIGH_FLOW_ALARM AND NOT "DB2120_MPP_ITC_IPC".RESET_FAULTS));
   #NOZZLE_FLOW_SETPOINT_ALARM := #_w1 AND ((#LASER_READY AND #NOZZLE_COOLING_TEMP_RAW_INPUT.%X0 AND #O_BYTE_0.NOZZLE_FLOW_ANALOG_VALUE) OR (#NOZZLE_FLOW_SETPOINT_ALARM AND NOT "DB2120_MPP_ITC_IPC".RESET_FAULTS));
END_REGION

REGION Network 9: COOLING SENSOR NOZZLE TEMPERATURE WARNINGS/ALARMS
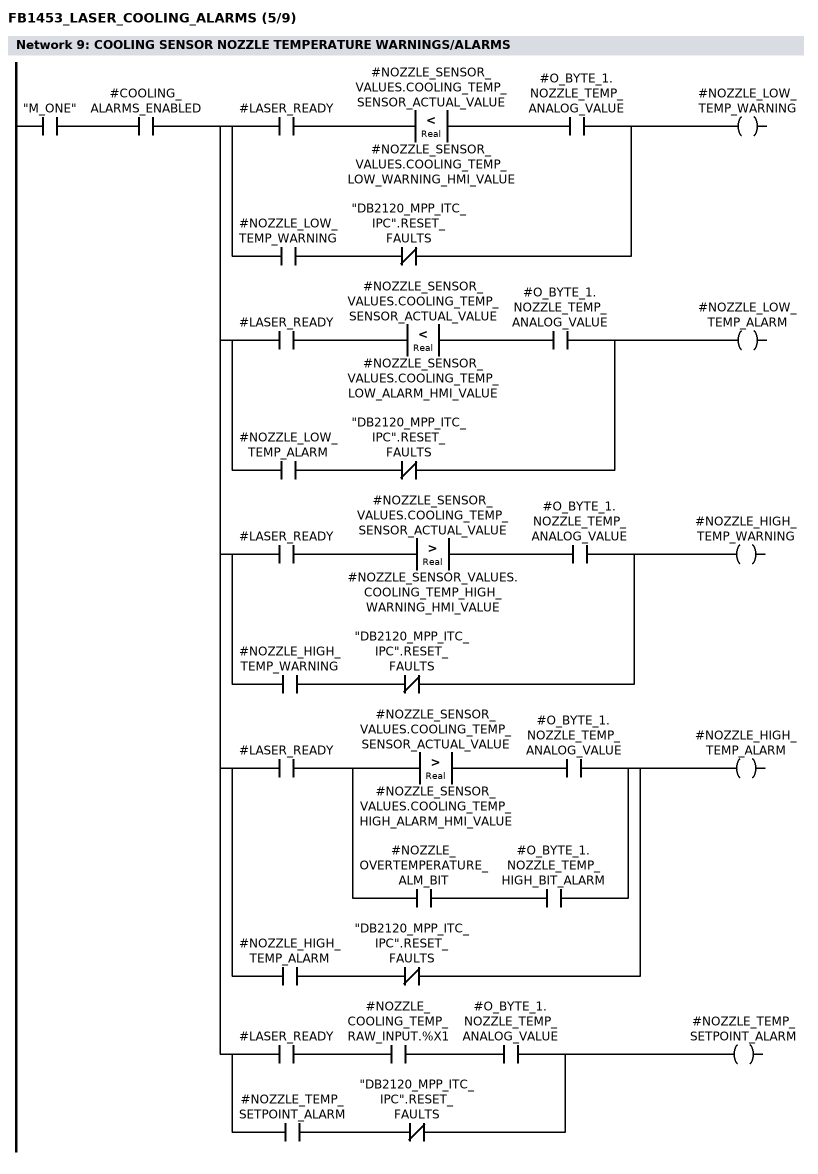
   RUNG wire#powerrail
      Contact( "M_ONE" )
      Contact( #COOLING_ALARMS_ENABLED )
      wire#w1
      Contact( #LASER_READY )
      { S7_Templates := "SrcType := Real" } LT_Contact(in1 := #NOZZLE_SENSOR_VALUES.COOLING_TEMP_SENSOR_ACTUAL_VALUE, in2 := #NOZZLE_SENSOR_VALUES.COOLING_TEMP_LOW_WARNING_HMI_VALUE)
      Contact( #O_BYTE_1.NOZZLE_TEMP_ANALOG_VALUE )
      wire#w2
      Coil( #NOZZLE_LOW_TEMP_WARNING )
   END_RUNG
   RUNG wire#w1
      Contact( #NOZZLE_LOW_TEMP_WARNING )
      I_Contact( "DB2120_MPP_ITC_IPC".RESET_FAULTS )
   END_RUNG wire#w2
   RUNG wire#w1
      Contact( #LASER_READY )
      { S7_Templates := "SrcType := Real" } LT_Contact(in1 := #NOZZLE_SENSOR_VALUES.COOLING_TEMP_SENSOR_ACTUAL_VALUE, in2 := #NOZZLE_SENSOR_VALUES.COOLING_TEMP_LOW_ALARM_HMI_VALUE)
      Contact( #O_BYTE_1.NOZZLE_TEMP_ANALOG_VALUE )
      wire#w3
      Coil( #NOZZLE_LOW_TEMP_ALARM )
   END_RUNG
   RUNG wire#w1
      Contact( #NOZZLE_LOW_TEMP_ALARM )
      I_Contact( "DB2120_MPP_ITC_IPC".RESET_FAULTS )
   END_RUNG wire#w3
   RUNG wire#w1
      Contact( #LASER_READY )
      { S7_Templates := "SrcType := Real" } GT_Contact(in1 := #NOZZLE_SENSOR_VALUES.COOLING_TEMP_SENSOR_ACTUAL_VALUE, in2 := #NOZZLE_SENSOR_VALUES.COOLING_TEMP_HIGH_WARNING_HMI_VALUE)
      Contact( #O_BYTE_1.NOZZLE_TEMP_ANALOG_VALUE )
      wire#w4
      Coil( #NOZZLE_HIGH_TEMP_WARNING )
   END_RUNG
   RUNG wire#w1
      Contact( #NOZZLE_HIGH_TEMP_WARNING )
      I_Contact( "DB2120_MPP_ITC_IPC".RESET_FAULTS )
   END_RUNG wire#w4
   RUNG wire#w1
      Contact( #LASER_READY )
      wire#w5
      { S7_Templates := "SrcType := Real" } GT_Contact(in1 := #NOZZLE_SENSOR_VALUES.COOLING_TEMP_SENSOR_ACTUAL_VALUE, in2 := #NOZZLE_SENSOR_VALUES.COOLING_TEMP_HIGH_ALARM_HMI_VALUE)
      Contact( #O_BYTE_1.NOZZLE_TEMP_ANALOG_VALUE )
      wire#w6
      Coil( #NOZZLE_HIGH_TEMP_ALARM )
   END_RUNG
   RUNG wire#w5
      Contact( #NOZZLE_OVERTEMPERATURE_ALM_BIT )
      Contact( #O_BYTE_1.NOZZLE_TEMP_HIGH_BIT_ALARM )
   END_RUNG wire#w6
   RUNG wire#w1
      Contact( #NOZZLE_HIGH_TEMP_ALARM )
      I_Contact( "DB2120_MPP_ITC_IPC".RESET_FAULTS )
   END_RUNG wire#w6
   RUNG wire#w1
      Contact( #LASER_READY )
      Contact( #NOZZLE_COOLING_TEMP_RAW_INPUT.%X1 )
      Contact( #O_BYTE_1.NOZZLE_TEMP_ANALOG_VALUE )
      wire#w7
      Coil( #NOZZLE_TEMP_SETPOINT_ALARM )
   END_RUNG
   RUNG wire#w1
      Contact( #NOZZLE_TEMP_SETPOINT_ALARM )
      I_Contact( "DB2120_MPP_ITC_IPC".RESET_FAULTS )
   END_RUNG wire#w7
   // the same network as SCL:
   #_w1 := "M_ONE" AND #COOLING_ALARMS_ENABLED;
   #NOZZLE_LOW_TEMP_WARNING := #_w1 AND ((#LASER_READY AND (#NOZZLE_SENSOR_VALUES.COOLING_TEMP_SENSOR_ACTUAL_VALUE < #NOZZLE_SENSOR_VALUES.COOLING_TEMP_LOW_WARNING_HMI_VALUE) AND #O_BYTE_1.NOZZLE_TEMP_ANALOG_VALUE) OR (#NOZZLE_LOW_TEMP_WARNING AND NOT "DB2120_MPP_ITC_IPC".RESET_FAULTS));
   #NOZZLE_LOW_TEMP_ALARM := #_w1 AND ((#LASER_READY AND (#NOZZLE_SENSOR_VALUES.COOLING_TEMP_SENSOR_ACTUAL_VALUE < #NOZZLE_SENSOR_VALUES.COOLING_TEMP_LOW_ALARM_HMI_VALUE) AND #O_BYTE_1.NOZZLE_TEMP_ANALOG_VALUE) OR (#NOZZLE_LOW_TEMP_ALARM AND NOT "DB2120_MPP_ITC_IPC".RESET_FAULTS));
   #NOZZLE_HIGH_TEMP_WARNING := #_w1 AND ((#LASER_READY AND (#NOZZLE_SENSOR_VALUES.COOLING_TEMP_SENSOR_ACTUAL_VALUE > #NOZZLE_SENSOR_VALUES.COOLING_TEMP_HIGH_WARNING_HMI_VALUE) AND #O_BYTE_1.NOZZLE_TEMP_ANALOG_VALUE) OR (#NOZZLE_HIGH_TEMP_WARNING AND NOT "DB2120_MPP_ITC_IPC".RESET_FAULTS));
   #NOZZLE_HIGH_TEMP_ALARM := #_w1 AND ((#LASER_READY AND (((#NOZZLE_SENSOR_VALUES.COOLING_TEMP_SENSOR_ACTUAL_VALUE > #NOZZLE_SENSOR_VALUES.COOLING_TEMP_HIGH_ALARM_HMI_VALUE) AND #O_BYTE_1.NOZZLE_TEMP_ANALOG_VALUE) OR (#NOZZLE_OVERTEMPERATURE_ALM_BIT AND #O_BYTE_1.NOZZLE_TEMP_HIGH_BIT_ALARM))) OR (#NOZZLE_HIGH_TEMP_ALARM AND NOT "DB2120_MPP_ITC_IPC".RESET_FAULTS));
   #NOZZLE_TEMP_SETPOINT_ALARM := #_w1 AND ((#LASER_READY AND #NOZZLE_COOLING_TEMP_RAW_INPUT.%X1 AND #O_BYTE_1.NOZZLE_TEMP_ANALOG_VALUE) OR (#NOZZLE_TEMP_SETPOINT_ALARM AND NOT "DB2120_MPP_ITC_IPC".RESET_FAULTS));
END_REGION

REGION Network 10: COOLING SENSOR LASER HEAD FLOW WARNINGS/ALARMS
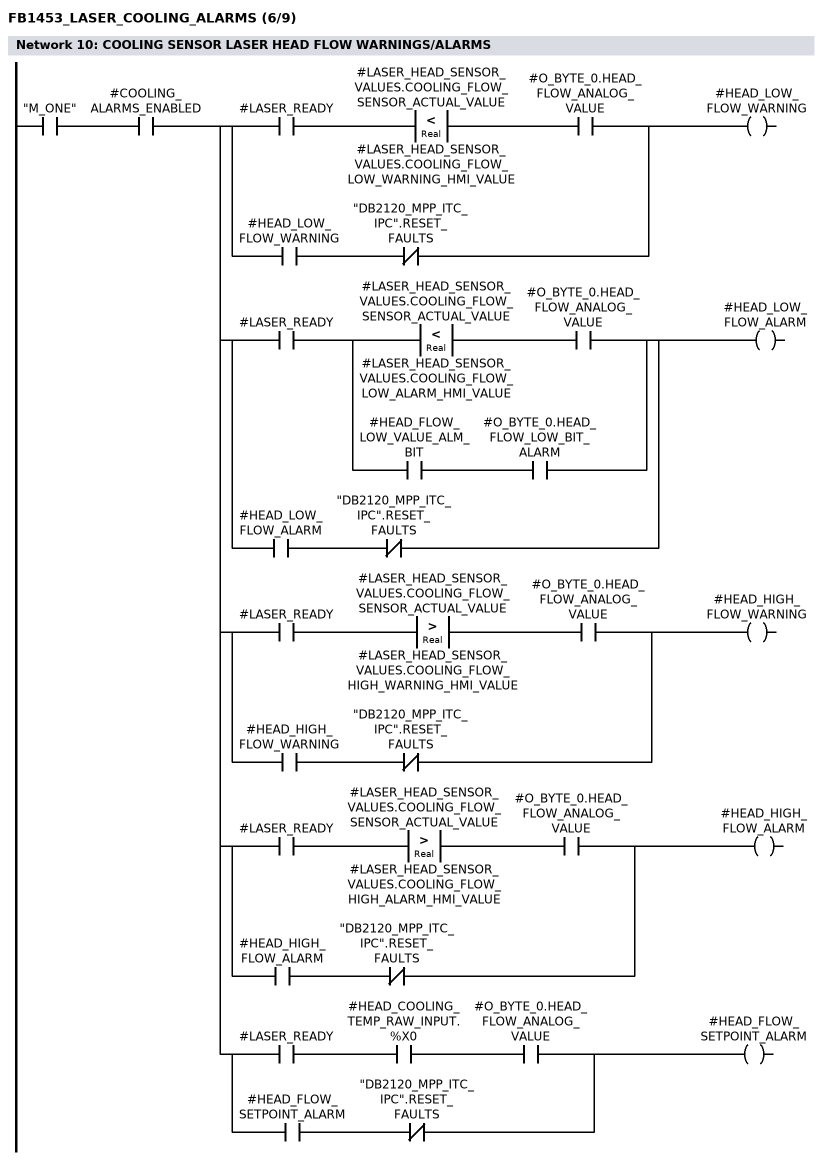
   RUNG wire#powerrail
      Contact( "M_ONE" )
      Contact( #COOLING_ALARMS_ENABLED )
      wire#w1
      Contact( #LASER_READY )
      { S7_Templates := "SrcType := Real" } LT_Contact(in1 := #LASER_HEAD_SENSOR_VALUES.COOLING_FLOW_SENSOR_ACTUAL_VALUE, in2 := #LASER_HEAD_SENSOR_VALUES.COOLING_FLOW_LOW_WARNING_HMI_VALUE)
      Contact( #O_BYTE_0.HEAD_FLOW_ANALOG_VALUE )
      wire#w2
      Coil( #HEAD_LOW_FLOW_WARNING )
   END_RUNG
   RUNG wire#w1
      Contact( #HEAD_LOW_FLOW_WARNING )
      I_Contact( "DB2120_MPP_ITC_IPC".RESET_FAULTS )
   END_RUNG wire#w2
   RUNG wire#w1
      Contact( #LASER_READY )
      wire#w3
      { S7_Templates := "SrcType := Real" } LT_Contact(in1 := #LASER_HEAD_SENSOR_VALUES.COOLING_FLOW_SENSOR_ACTUAL_VALUE, in2 := #LASER_HEAD_SENSOR_VALUES.COOLING_FLOW_LOW_ALARM_HMI_VALUE)
      Contact( #O_BYTE_0.HEAD_FLOW_ANALOG_VALUE )
      wire#w4
      Coil( #HEAD_LOW_FLOW_ALARM )
   END_RUNG
   RUNG wire#w3
      Contact( #HEAD_FLOW_LOW_VALUE_ALM_BIT )
      Contact( #O_BYTE_0.HEAD_FLOW_LOW_BIT_ALARM )
   END_RUNG wire#w4
   RUNG wire#w1
      Contact( #HEAD_LOW_FLOW_ALARM )
      I_Contact( "DB2120_MPP_ITC_IPC".RESET_FAULTS )
   END_RUNG wire#w4
   RUNG wire#w1
      Contact( #LASER_READY )
      { S7_Templates := "SrcType := Real" } GT_Contact(in1 := #LASER_HEAD_SENSOR_VALUES.COOLING_FLOW_SENSOR_ACTUAL_VALUE, in2 := #LASER_HEAD_SENSOR_VALUES.COOLING_FLOW_HIGH_WARNING_HMI_VALUE)
      Contact( #O_BYTE_0.HEAD_FLOW_ANALOG_VALUE )
      wire#w5
      Coil( #HEAD_HIGH_FLOW_WARNING )
   END_RUNG
   RUNG wire#w1
      Contact( #HEAD_HIGH_FLOW_WARNING )
      I_Contact( "DB2120_MPP_ITC_IPC".RESET_FAULTS )
   END_RUNG wire#w5
   RUNG wire#w1
      Contact( #LASER_READY )
      { S7_Templates := "SrcType := Real" } GT_Contact(in1 := #LASER_HEAD_SENSOR_VALUES.COOLING_FLOW_SENSOR_ACTUAL_VALUE, in2 := #LASER_HEAD_SENSOR_VALUES.COOLING_FLOW_HIGH_ALARM_HMI_VALUE)
      Contact( #O_BYTE_0.HEAD_FLOW_ANALOG_VALUE )
      wire#w6
      Coil( #HEAD_HIGH_FLOW_ALARM )
   END_RUNG
   RUNG wire#w1
      Contact( #HEAD_HIGH_FLOW_ALARM )
      I_Contact( "DB2120_MPP_ITC_IPC".RESET_FAULTS )
   END_RUNG wire#w6
   RUNG wire#w1
      Contact( #LASER_READY )
      Contact( #HEAD_COOLING_TEMP_RAW_INPUT.%X0 )
      Contact( #O_BYTE_0.HEAD_FLOW_ANALOG_VALUE )
      wire#w7
      Coil( #HEAD_FLOW_SETPOINT_ALARM )
   END_RUNG
   RUNG wire#w1
      Contact( #HEAD_FLOW_SETPOINT_ALARM )
      I_Contact( "DB2120_MPP_ITC_IPC".RESET_FAULTS )
   END_RUNG wire#w7
   // the same network as SCL:
   #_w1 := "M_ONE" AND #COOLING_ALARMS_ENABLED;
   #HEAD_LOW_FLOW_WARNING := #_w1 AND ((#LASER_READY AND (#LASER_HEAD_SENSOR_VALUES.COOLING_FLOW_SENSOR_ACTUAL_VALUE < #LASER_HEAD_SENSOR_VALUES.COOLING_FLOW_LOW_WARNING_HMI_VALUE) AND #O_BYTE_0.HEAD_FLOW_ANALOG_VALUE) OR (#HEAD_LOW_FLOW_WARNING AND NOT "DB2120_MPP_ITC_IPC".RESET_FAULTS));
   #HEAD_LOW_FLOW_ALARM := #_w1 AND ((#LASER_READY AND (((#LASER_HEAD_SENSOR_VALUES.COOLING_FLOW_SENSOR_ACTUAL_VALUE < #LASER_HEAD_SENSOR_VALUES.COOLING_FLOW_LOW_ALARM_HMI_VALUE) AND #O_BYTE_0.HEAD_FLOW_ANALOG_VALUE) OR (#HEAD_FLOW_LOW_VALUE_ALM_BIT AND #O_BYTE_0.HEAD_FLOW_LOW_BIT_ALARM))) OR (#HEAD_LOW_FLOW_ALARM AND NOT "DB2120_MPP_ITC_IPC".RESET_FAULTS));
   #HEAD_HIGH_FLOW_WARNING := #_w1 AND ((#LASER_READY AND (#LASER_HEAD_SENSOR_VALUES.COOLING_FLOW_SENSOR_ACTUAL_VALUE > #LASER_HEAD_SENSOR_VALUES.COOLING_FLOW_HIGH_WARNING_HMI_VALUE) AND #O_BYTE_0.HEAD_FLOW_ANALOG_VALUE) OR (#HEAD_HIGH_FLOW_WARNING AND NOT "DB2120_MPP_ITC_IPC".RESET_FAULTS));
   #HEAD_HIGH_FLOW_ALARM := #_w1 AND ((#LASER_READY AND (#LASER_HEAD_SENSOR_VALUES.COOLING_FLOW_SENSOR_ACTUAL_VALUE > #LASER_HEAD_SENSOR_VALUES.COOLING_FLOW_HIGH_ALARM_HMI_VALUE) AND #O_BYTE_0.HEAD_FLOW_ANALOG_VALUE) OR (#HEAD_HIGH_FLOW_ALARM AND NOT "DB2120_MPP_ITC_IPC".RESET_FAULTS));
   #HEAD_FLOW_SETPOINT_ALARM := #_w1 AND ((#LASER_READY AND #HEAD_COOLING_TEMP_RAW_INPUT.%X0 AND #O_BYTE_0.HEAD_FLOW_ANALOG_VALUE) OR (#HEAD_FLOW_SETPOINT_ALARM AND NOT "DB2120_MPP_ITC_IPC".RESET_FAULTS));
END_REGION

REGION Network 11: COOLING SENSOR LASER HEAD TEMPERATURE WARNINGS/ALARMS
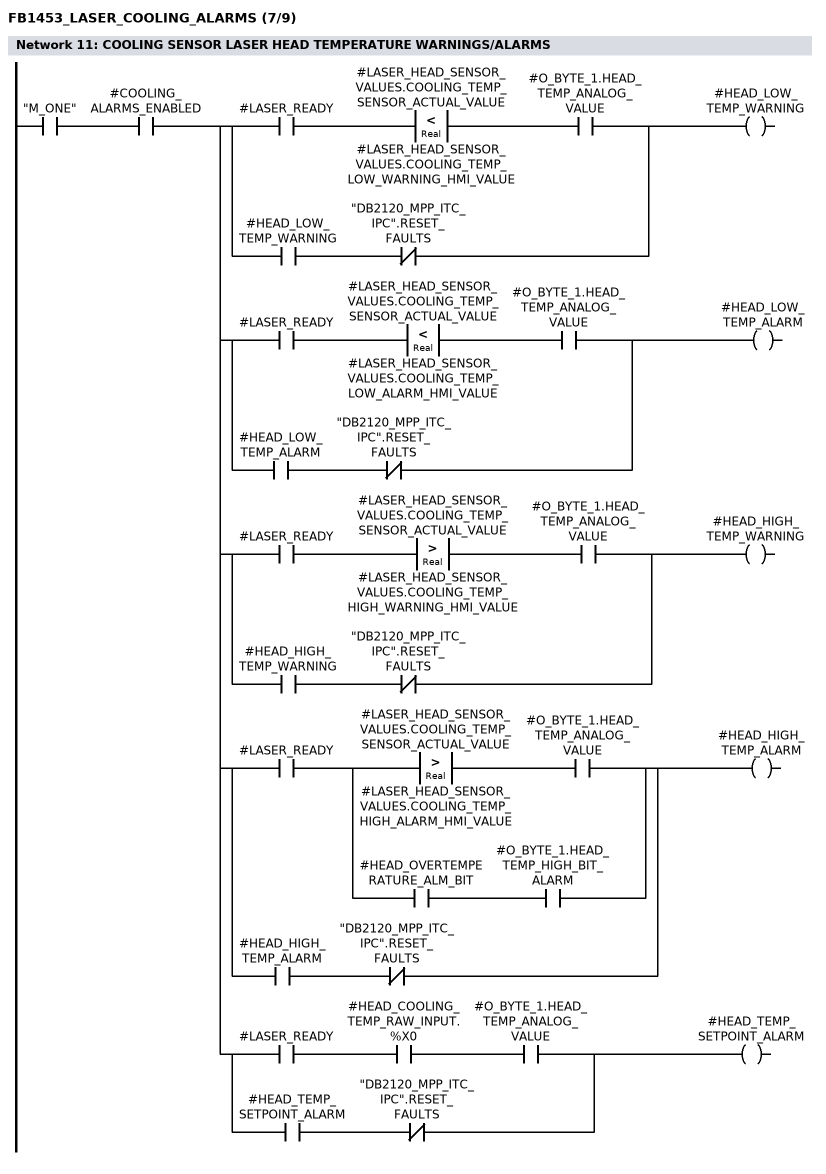
   RUNG wire#powerrail
      Contact( "M_ONE" )
      Contact( #COOLING_ALARMS_ENABLED )
      wire#w1
      Contact( #LASER_READY )
      { S7_Templates := "SrcType := Real" } LT_Contact(in1 := #LASER_HEAD_SENSOR_VALUES.COOLING_TEMP_SENSOR_ACTUAL_VALUE, in2 := #LASER_HEAD_SENSOR_VALUES.COOLING_TEMP_LOW_WARNING_HMI_VALUE)
      Contact( #O_BYTE_1.HEAD_TEMP_ANALOG_VALUE )
      wire#w2
      Coil( #HEAD_LOW_TEMP_WARNING )
   END_RUNG
   RUNG wire#w1
      Contact( #HEAD_LOW_TEMP_WARNING )
      I_Contact( "DB2120_MPP_ITC_IPC".RESET_FAULTS )
   END_RUNG wire#w2
   RUNG wire#w1
      Contact( #LASER_READY )
      { S7_Templates := "SrcType := Real" } LT_Contact(in1 := #LASER_HEAD_SENSOR_VALUES.COOLING_TEMP_SENSOR_ACTUAL_VALUE, in2 := #LASER_HEAD_SENSOR_VALUES.COOLING_TEMP_LOW_ALARM_HMI_VALUE)
      Contact( #O_BYTE_1.HEAD_TEMP_ANALOG_VALUE )
      wire#w3
      Coil( #HEAD_LOW_TEMP_ALARM )
   END_RUNG
   RUNG wire#w1
      Contact( #HEAD_LOW_TEMP_ALARM )
      I_Contact( "DB2120_MPP_ITC_IPC".RESET_FAULTS )
   END_RUNG wire#w3
   RUNG wire#w1
      Contact( #LASER_READY )
      { S7_Templates := "SrcType := Real" } GT_Contact(in1 := #LASER_HEAD_SENSOR_VALUES.COOLING_TEMP_SENSOR_ACTUAL_VALUE, in2 := #LASER_HEAD_SENSOR_VALUES.COOLING_TEMP_HIGH_WARNING_HMI_VALUE)
      Contact( #O_BYTE_1.HEAD_TEMP_ANALOG_VALUE )
      wire#w4
      Coil( #HEAD_HIGH_TEMP_WARNING )
   END_RUNG
   RUNG wire#w1
      Contact( #HEAD_HIGH_TEMP_WARNING )
      I_Contact( "DB2120_MPP_ITC_IPC".RESET_FAULTS )
   END_RUNG wire#w4
   RUNG wire#w1
      Contact( #LASER_READY )
      wire#w5
      { S7_Templates := "SrcType := Real" } GT_Contact(in1 := #LASER_HEAD_SENSOR_VALUES.COOLING_TEMP_SENSOR_ACTUAL_VALUE, in2 := #LASER_HEAD_SENSOR_VALUES.COOLING_TEMP_HIGH_ALARM_HMI_VALUE)
      Contact( #O_BYTE_1.HEAD_TEMP_ANALOG_VALUE )
      wire#w6
      Coil( #HEAD_HIGH_TEMP_ALARM )
   END_RUNG
   RUNG wire#w5
      Contact( #HEAD_OVERTEMPERATURE_ALM_BIT )
      Contact( #O_BYTE_1.HEAD_TEMP_HIGH_BIT_ALARM )
   END_RUNG wire#w6
   RUNG wire#w1
      Contact( #HEAD_HIGH_TEMP_ALARM )
      I_Contact( "DB2120_MPP_ITC_IPC".RESET_FAULTS )
   END_RUNG wire#w6
   RUNG wire#w1
      Contact( #LASER_READY )
      Contact( #HEAD_COOLING_TEMP_RAW_INPUT.%X0 )
      Contact( #O_BYTE_1.HEAD_TEMP_ANALOG_VALUE )
      wire#w7
      Coil( #HEAD_TEMP_SETPOINT_ALARM )
   END_RUNG
   RUNG wire#w1
      Contact( #HEAD_TEMP_SETPOINT_ALARM )
      I_Contact( "DB2120_MPP_ITC_IPC".RESET_FAULTS )
   END_RUNG wire#w7
   // the same network as SCL:
   #_w1 := "M_ONE" AND #COOLING_ALARMS_ENABLED;
   #HEAD_LOW_TEMP_WARNING := #_w1 AND ((#LASER_READY AND (#LASER_HEAD_SENSOR_VALUES.COOLING_TEMP_SENSOR_ACTUAL_VALUE < #LASER_HEAD_SENSOR_VALUES.COOLING_TEMP_LOW_WARNING_HMI_VALUE) AND #O_BYTE_1.HEAD_TEMP_ANALOG_VALUE) OR (#HEAD_LOW_TEMP_WARNING AND NOT "DB2120_MPP_ITC_IPC".RESET_FAULTS));
   #HEAD_LOW_TEMP_ALARM := #_w1 AND ((#LASER_READY AND (#LASER_HEAD_SENSOR_VALUES.COOLING_TEMP_SENSOR_ACTUAL_VALUE < #LASER_HEAD_SENSOR_VALUES.COOLING_TEMP_LOW_ALARM_HMI_VALUE) AND #O_BYTE_1.HEAD_TEMP_ANALOG_VALUE) OR (#HEAD_LOW_TEMP_ALARM AND NOT "DB2120_MPP_ITC_IPC".RESET_FAULTS));
   #HEAD_HIGH_TEMP_WARNING := #_w1 AND ((#LASER_READY AND (#LASER_HEAD_SENSOR_VALUES.COOLING_TEMP_SENSOR_ACTUAL_VALUE > #LASER_HEAD_SENSOR_VALUES.COOLING_TEMP_HIGH_WARNING_HMI_VALUE) AND #O_BYTE_1.HEAD_TEMP_ANALOG_VALUE) OR (#HEAD_HIGH_TEMP_WARNING AND NOT "DB2120_MPP_ITC_IPC".RESET_FAULTS));
   #HEAD_HIGH_TEMP_ALARM := #_w1 AND ((#LASER_READY AND (((#LASER_HEAD_SENSOR_VALUES.COOLING_TEMP_SENSOR_ACTUAL_VALUE > #LASER_HEAD_SENSOR_VALUES.COOLING_TEMP_HIGH_ALARM_HMI_VALUE) AND #O_BYTE_1.HEAD_TEMP_ANALOG_VALUE) OR (#HEAD_OVERTEMPERATURE_ALM_BIT AND #O_BYTE_1.HEAD_TEMP_HIGH_BIT_ALARM))) OR (#HEAD_HIGH_TEMP_ALARM AND NOT "DB2120_MPP_ITC_IPC".RESET_FAULTS));
   #HEAD_TEMP_SETPOINT_ALARM := #_w1 AND ((#LASER_READY AND #HEAD_COOLING_TEMP_RAW_INPUT.%X0 AND #O_BYTE_1.HEAD_TEMP_ANALOG_VALUE) OR (#HEAD_TEMP_SETPOINT_ALARM AND NOT "DB2120_MPP_ITC_IPC".RESET_FAULTS));
END_REGION

REGION Network 12: INMEDIATE AND STOP END OF CYCLE ALARMS
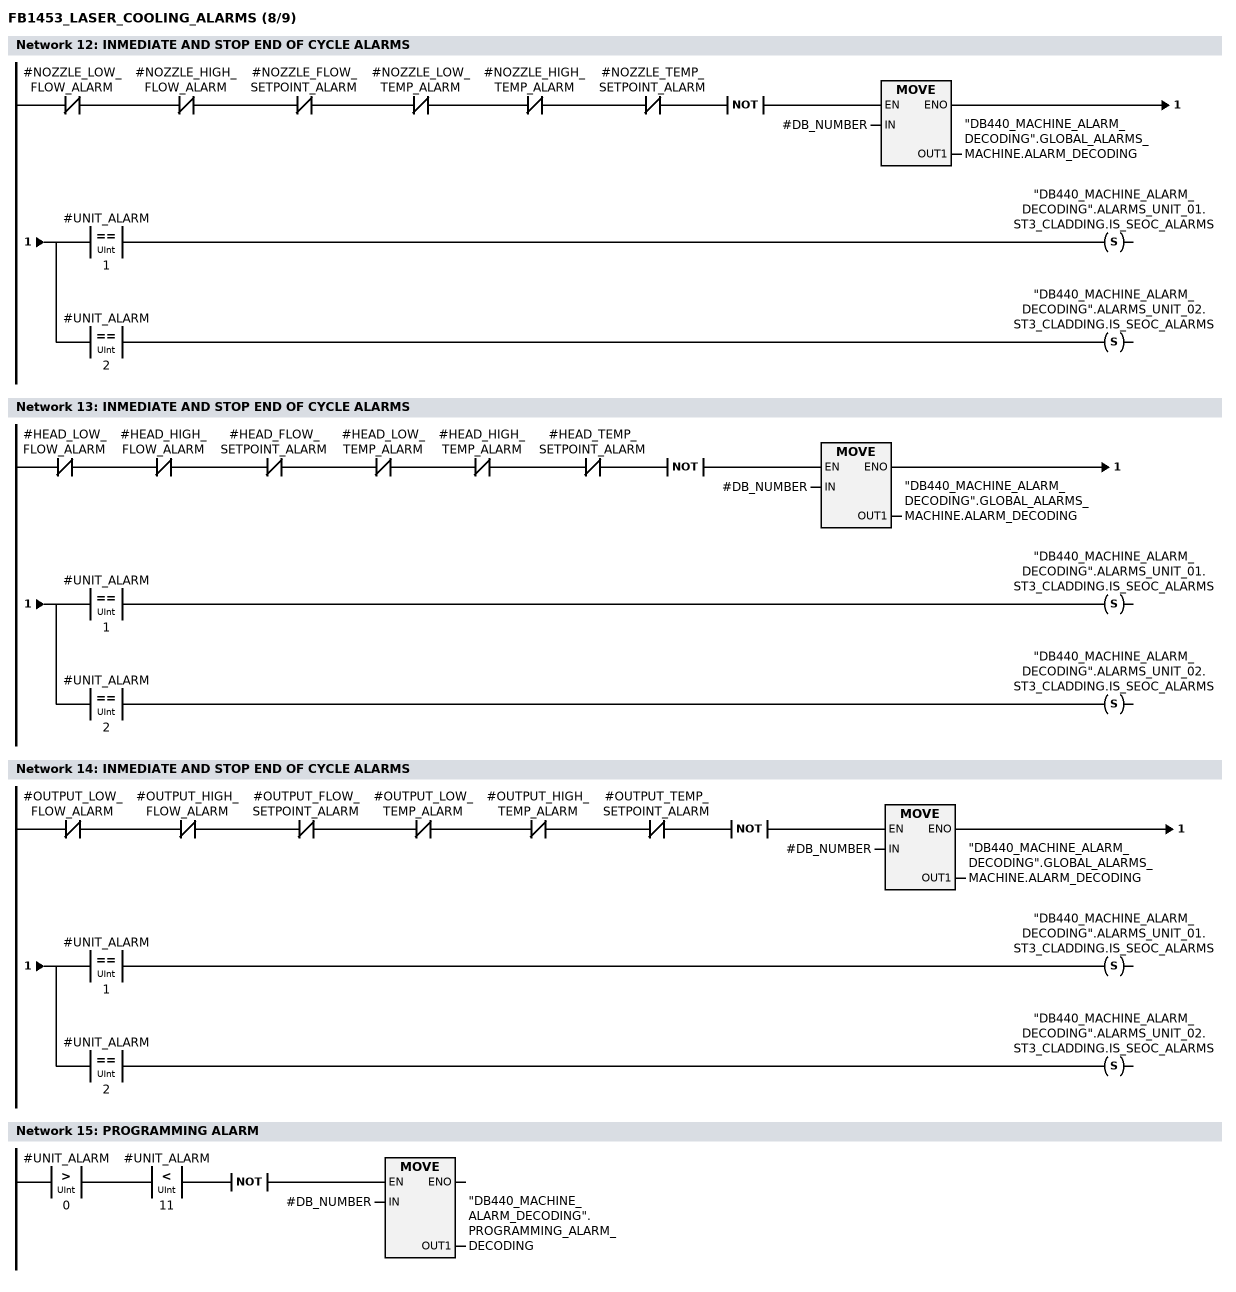
   RUNG wire#powerrail
      I_Contact( #NOZZLE_LOW_FLOW_ALARM )
      I_Contact( #NOZZLE_HIGH_FLOW_ALARM )
      I_Contact( #NOZZLE_FLOW_SETPOINT_ALARM )
      I_Contact( #NOZZLE_LOW_TEMP_ALARM )
      I_Contact( #NOZZLE_HIGH_TEMP_ALARM )
      I_Contact( #NOZZLE_TEMP_SETPOINT_ALARM )
      Not()
      { S7_GenerateENO := "TRUE" } Move(in := #DB_NUMBER, out1 => "DB440_MACHINE_ALARM_DECODING".GLOBAL_ALARMS_MACHINE.ALARM_DECODING)
      wire#w1
      { S7_Templates := "SrcType := UInt" } EQ_Contact(in1 := #UNIT_ALARM, in2 := 1)
      S_Coil( "DB440_MACHINE_ALARM_DECODING".ALARMS_UNIT_01.ST3_CLADDING.IS_SEOC_ALARMS )
   END_RUNG
   RUNG wire#w1
      { S7_Templates := "SrcType := UInt" } EQ_Contact(in1 := #UNIT_ALARM, in2 := 2)
      S_Coil( "DB440_MACHINE_ALARM_DECODING".ALARMS_UNIT_02.ST3_CLADDING.IS_SEOC_ALARMS )
   END_RUNG
   // the same network as SCL:
   // ENO of a box is taken as its EN; it also drops when the box reports an error
   #_w1 := NOT (NOT #NOZZLE_LOW_FLOW_ALARM AND NOT #NOZZLE_HIGH_FLOW_ALARM AND NOT #NOZZLE_FLOW_SETPOINT_ALARM AND NOT #NOZZLE_LOW_TEMP_ALARM AND NOT #NOZZLE_HIGH_TEMP_ALARM AND NOT #NOZZLE_TEMP_SETPOINT_ALARM);
   IF #_w1 THEN "DB440_MACHINE_ALARM_DECODING".GLOBAL_ALARMS_MACHINE.ALARM_DECODING := #DB_NUMBER; END_IF;
   IF #_w1 AND (#UNIT_ALARM = 1) THEN
       "DB440_MACHINE_ALARM_DECODING".ALARMS_UNIT_01.ST3_CLADDING.IS_SEOC_ALARMS := TRUE;
   END_IF;
   IF #_w1 AND (#UNIT_ALARM = 2) THEN
       "DB440_MACHINE_ALARM_DECODING".ALARMS_UNIT_02.ST3_CLADDING.IS_SEOC_ALARMS := TRUE;
   END_IF;
END_REGION

REGION Network 13: INMEDIATE AND STOP END OF CYCLE ALARMS
   RUNG wire#powerrail
      I_Contact( #HEAD_LOW_FLOW_ALARM )
      I_Contact( #HEAD_HIGH_FLOW_ALARM )
      I_Contact( #HEAD_FLOW_SETPOINT_ALARM )
      I_Contact( #HEAD_LOW_TEMP_ALARM )
      I_Contact( #HEAD_HIGH_TEMP_ALARM )
      I_Contact( #HEAD_TEMP_SETPOINT_ALARM )
      Not()
      { S7_GenerateENO := "TRUE" } Move(in := #DB_NUMBER, out1 => "DB440_MACHINE_ALARM_DECODING".GLOBAL_ALARMS_MACHINE.ALARM_DECODING)
      wire#w1
      { S7_Templates := "SrcType := UInt" } EQ_Contact(in1 := #UNIT_ALARM, in2 := 1)
      S_Coil( "DB440_MACHINE_ALARM_DECODING".ALARMS_UNIT_01.ST3_CLADDING.IS_SEOC_ALARMS )
   END_RUNG
   RUNG wire#w1
      { S7_Templates := "SrcType := UInt" } EQ_Contact(in1 := #UNIT_ALARM, in2 := 2)
      S_Coil( "DB440_MACHINE_ALARM_DECODING".ALARMS_UNIT_02.ST3_CLADDING.IS_SEOC_ALARMS )
   END_RUNG
   // the same network as SCL:
   // ENO of a box is taken as its EN; it also drops when the box reports an error
   #_w1 := NOT (NOT #HEAD_LOW_FLOW_ALARM AND NOT #HEAD_HIGH_FLOW_ALARM AND NOT #HEAD_FLOW_SETPOINT_ALARM AND NOT #HEAD_LOW_TEMP_ALARM AND NOT #HEAD_HIGH_TEMP_ALARM AND NOT #HEAD_TEMP_SETPOINT_ALARM);
   IF #_w1 THEN "DB440_MACHINE_ALARM_DECODING".GLOBAL_ALARMS_MACHINE.ALARM_DECODING := #DB_NUMBER; END_IF;
   IF #_w1 AND (#UNIT_ALARM = 1) THEN
       "DB440_MACHINE_ALARM_DECODING".ALARMS_UNIT_01.ST3_CLADDING.IS_SEOC_ALARMS := TRUE;
   END_IF;
   IF #_w1 AND (#UNIT_ALARM = 2) THEN
       "DB440_MACHINE_ALARM_DECODING".ALARMS_UNIT_02.ST3_CLADDING.IS_SEOC_ALARMS := TRUE;
   END_IF;
END_REGION

REGION Network 14: INMEDIATE AND STOP END OF CYCLE ALARMS
   RUNG wire#powerrail
      I_Contact( #OUTPUT_LOW_FLOW_ALARM )
      I_Contact( #OUTPUT_HIGH_FLOW_ALARM )
      I_Contact( #OUTPUT_FLOW_SETPOINT_ALARM )
      I_Contact( #OUTPUT_LOW_TEMP_ALARM )
      I_Contact( #OUTPUT_HIGH_TEMP_ALARM )
      I_Contact( #OUTPUT_TEMP_SETPOINT_ALARM )
      Not()
      { S7_GenerateENO := "TRUE" } Move(in := #DB_NUMBER, out1 => "DB440_MACHINE_ALARM_DECODING".GLOBAL_ALARMS_MACHINE.ALARM_DECODING)
      wire#w1
      { S7_Templates := "SrcType := UInt" } EQ_Contact(in1 := #UNIT_ALARM, in2 := 1)
      S_Coil( "DB440_MACHINE_ALARM_DECODING".ALARMS_UNIT_01.ST3_CLADDING.IS_SEOC_ALARMS )
   END_RUNG
   RUNG wire#w1
      { S7_Templates := "SrcType := UInt" } EQ_Contact(in1 := #UNIT_ALARM, in2 := 2)
      S_Coil( "DB440_MACHINE_ALARM_DECODING".ALARMS_UNIT_02.ST3_CLADDING.IS_SEOC_ALARMS )
   END_RUNG
   // the same network as SCL:
   // ENO of a box is taken as its EN; it also drops when the box reports an error
   #_w1 := NOT (NOT #OUTPUT_LOW_FLOW_ALARM AND NOT #OUTPUT_HIGH_FLOW_ALARM AND NOT #OUTPUT_FLOW_SETPOINT_ALARM AND NOT #OUTPUT_LOW_TEMP_ALARM AND NOT #OUTPUT_HIGH_TEMP_ALARM AND NOT #OUTPUT_TEMP_SETPOINT_ALARM);
   IF #_w1 THEN "DB440_MACHINE_ALARM_DECODING".GLOBAL_ALARMS_MACHINE.ALARM_DECODING := #DB_NUMBER; END_IF;
   IF #_w1 AND (#UNIT_ALARM = 1) THEN
       "DB440_MACHINE_ALARM_DECODING".ALARMS_UNIT_01.ST3_CLADDING.IS_SEOC_ALARMS := TRUE;
   END_IF;
   IF #_w1 AND (#UNIT_ALARM = 2) THEN
       "DB440_MACHINE_ALARM_DECODING".ALARMS_UNIT_02.ST3_CLADDING.IS_SEOC_ALARMS := TRUE;
   END_IF;
END_REGION

REGION Network 15: PROGRAMMING ALARM
   RUNG wire#powerrail
      { S7_Templates := "SrcType := UInt" } GT_Contact(in1 := #UNIT_ALARM, in2 := 0)
      { S7_Templates := "SrcType := UInt" } LT_Contact(in1 := #UNIT_ALARM, in2 := 11)
      Not()
      Move(in := #DB_NUMBER, out1 => "DB440_MACHINE_ALARM_DECODING".PROGRAMMING_ALARM_DECODING)
   END_RUNG
   // the same network as SCL:
   IF NOT ((#UNIT_ALARM > 0) AND (#UNIT_ALARM < 11)) THEN
       "DB440_MACHINE_ALARM_DECODING".PROGRAMMING_ALARM_DECODING := #DB_NUMBER;
   END_IF;
END_REGION

REGION Network 16: WARNINGS
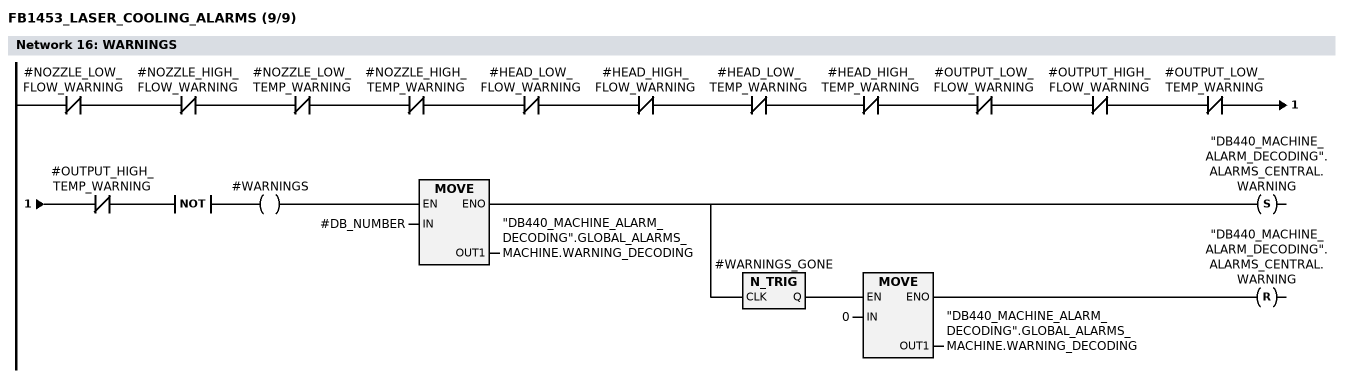
   RUNG wire#powerrail
      I_Contact( #NOZZLE_LOW_FLOW_WARNING )
      I_Contact( #NOZZLE_HIGH_FLOW_WARNING )
      I_Contact( #NOZZLE_LOW_TEMP_WARNING )
      I_Contact( #NOZZLE_HIGH_TEMP_WARNING )
      I_Contact( #HEAD_LOW_FLOW_WARNING )
      I_Contact( #HEAD_HIGH_FLOW_WARNING )
      I_Contact( #HEAD_LOW_TEMP_WARNING )
      I_Contact( #HEAD_HIGH_TEMP_WARNING )
      I_Contact( #OUTPUT_LOW_FLOW_WARNING )
      I_Contact( #OUTPUT_HIGH_FLOW_WARNING )
      I_Contact( #OUTPUT_LOW_TEMP_WARNING )
      I_Contact( #OUTPUT_HIGH_TEMP_WARNING )
      Not()
      Coil( #WARNINGS )
      Move(in := #DB_NUMBER, out1 => "DB440_MACHINE_ALARM_DECODING".GLOBAL_ALARMS_MACHINE.WARNING_DECODING)
      wire#w1
      S_Coil( "DB440_MACHINE_ALARM_DECODING".ALARMS_CENTRAL.WARNING )
   END_RUNG
   RUNG wire#w1
      N_Trig( #WARNINGS_GONE )
      Move(in := 0, out1 => "DB440_MACHINE_ALARM_DECODING".GLOBAL_ALARMS_MACHINE.WARNING_DECODING)
      R_Coil( "DB440_MACHINE_ALARM_DECODING".ALARMS_CENTRAL.WARNING )
   END_RUNG
   // the same network as SCL:
   #WARNINGS := NOT (NOT #NOZZLE_LOW_FLOW_WARNING AND NOT #NOZZLE_HIGH_FLOW_WARNING AND NOT #NOZZLE_LOW_TEMP_WARNING AND NOT #NOZZLE_HIGH_TEMP_WARNING AND NOT #HEAD_LOW_FLOW_WARNING AND NOT #HEAD_HIGH_FLOW_WARNING AND NOT #HEAD_LOW_TEMP_WARNING AND NOT #HEAD_HIGH_TEMP_WARNING AND NOT #OUTPUT_LOW_FLOW_WARNING AND NOT #OUTPUT_HIGH_FLOW_WARNING AND NOT #OUTPUT_LOW_TEMP_WARNING AND NOT #OUTPUT_HIGH_TEMP_WARNING);
   IF #WARNINGS THEN
       "DB440_MACHINE_ALARM_DECODING".GLOBAL_ALARMS_MACHINE.WARNING_DECODING := #DB_NUMBER;
       "DB440_MACHINE_ALARM_DECODING".ALARMS_CENTRAL.WARNING := TRUE;
   END_IF;
   #_w1 := NOT #WARNINGS AND #WARNINGS_GONE;   // falling edge
   #WARNINGS_GONE := #WARNINGS;
   IF #_w1 THEN
       "DB440_MACHINE_ALARM_DECODING".GLOBAL_ALARMS_MACHINE.WARNING_DECODING := 0;
       "DB440_MACHINE_ALARM_DECODING".ALARMS_CENTRAL.WARNING := FALSE;
   END_IF;
END_REGION
END_FUNCTION_BLOCK
